RoboDK station: ur10实机仿真.rdk

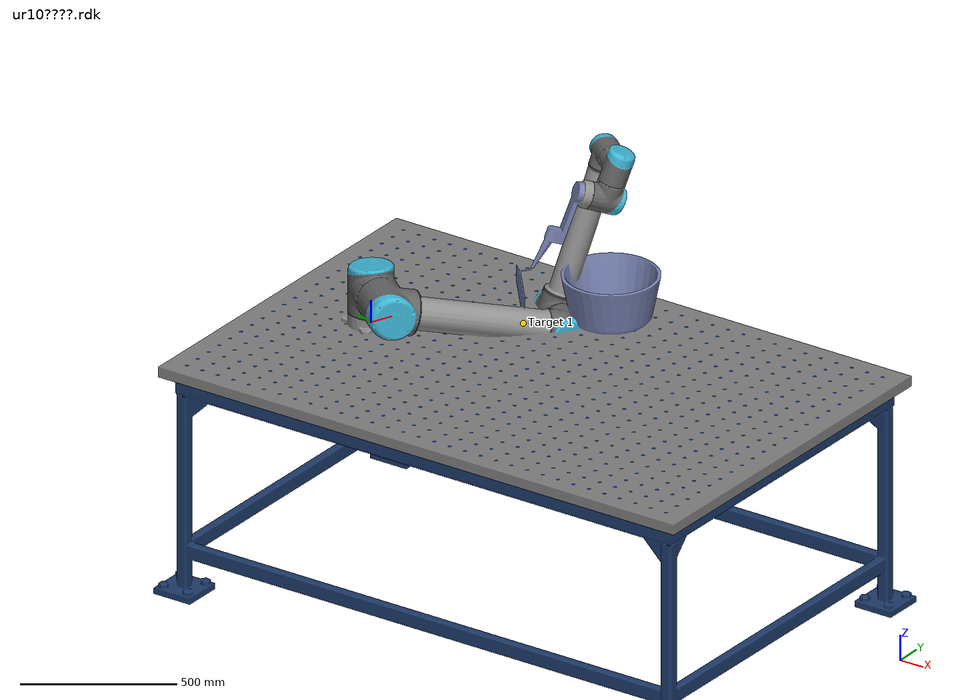
[picture v0: the station drawn from its stored meshes, robots at their saved joint values, targets as dots, program paths as lines]
Station ur10实机仿真 (saved by RoboDK 5.9.0). Poses are relative to the parent item; angles as X-Y-Z fixed-axis rotations.
  - object Table 2000x1200x800mm at (0, 0, 0) mm, size 2020 x 1340 x 800 mm, geometry from Table-2000x1200x800mm.sld
  - frame 工作坐标系 at (0, -9.36, 0) mm, rotated rx 0 ry 0 rz 68.84 deg
    - robot UR10: 6 axes, payload 10 kg, reach 1300 mm, repeatability 0.1 mm, weight 28.9 kg
        modified DH rows (alpha deg, a mm, theta deg, d mm): 0, 0, 0, 128; 90, 0, 180, 0; 0, 612.7, 0, 0; 0, 571.6, 0, 163.9; -90, 0, 0, 115.7; 90, 0, 180, 92.2
        joint limits [-360, -360, -360, -360, -360, -360] to [360, 360, 360, 360, 360, 360]; home [0, -90, -90, 0, 90, 0]; saved at [-17.375, -194.087, -273.743, 87.806, 92.707, -0.986]
      - tool , TCP at (-7.41, -480.84, 17.52) mm, rotated rx 110 ry 0 rz 0 deg, size 107.3 x 139.9 x 517.7 mm, geometry from .STEP
    - target Target 1 (Cartesian target) at (398.99, -274.73, 0) mm, rotated rx -180 ry 0 rz -110.26 deg; joints [-14.775, -88.651, -143.008, -38.34, 90, 5.481] of UR10
  - object  at (610, 450, 10) mm, rotated rx 90 ry 0 rz 0 deg, size 319.6 x 160 x 319.6 mm, geometry from .STEP
